// Mitsubishi GX Works2 project: Ex05   PLC: Q02/Q02H

PROGRAM MAIN
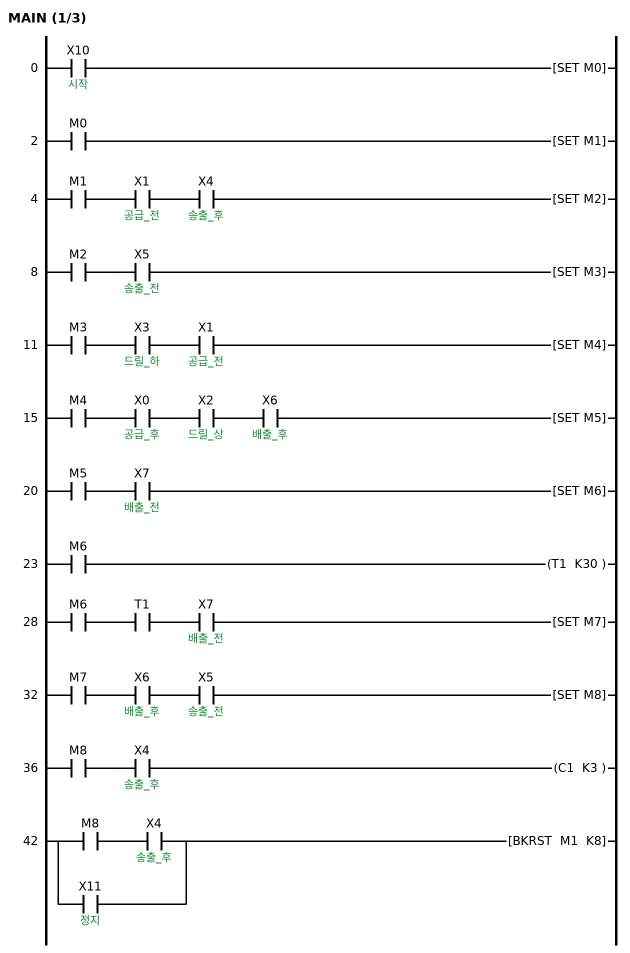
0     LD      X10  ; 시작
      SET     M0
2     LD      M0
      SET     M1
4     LD      M1
      AND     X1  ; 공급_전
      AND     X4  ; 송출_후
      SET     M2
8     LD      M2
      AND     X5  ; 송출_전
      SET     M3
11    LD      M3
      AND     X3  ; 드릴_하
      AND     X1  ; 공급_전
      SET     M4
15    LD      M4
      AND     X0  ; 공급_후
      AND     X2  ; 드릴_상
      AND     X6  ; 배출_후
      SET     M5
20    LD      M5
      AND     X7  ; 배출_전
      SET     M6
23    LD      M6
      OUT     T1 K30
28    LD      M6
      AND     T1
      AND     X7  ; 배출_전
      SET     M7
32    LD      M7
      AND     X6  ; 배출_후
      AND     X5  ; 송출_전
      SET     M8
36    LD      M8
      AND     X4  ; 송출_후
      OUT     C1 K3
42    LD      M8
      AND     X4  ; 송출_후
      OR      X11  ; 정지
      BKRST   M1 K8
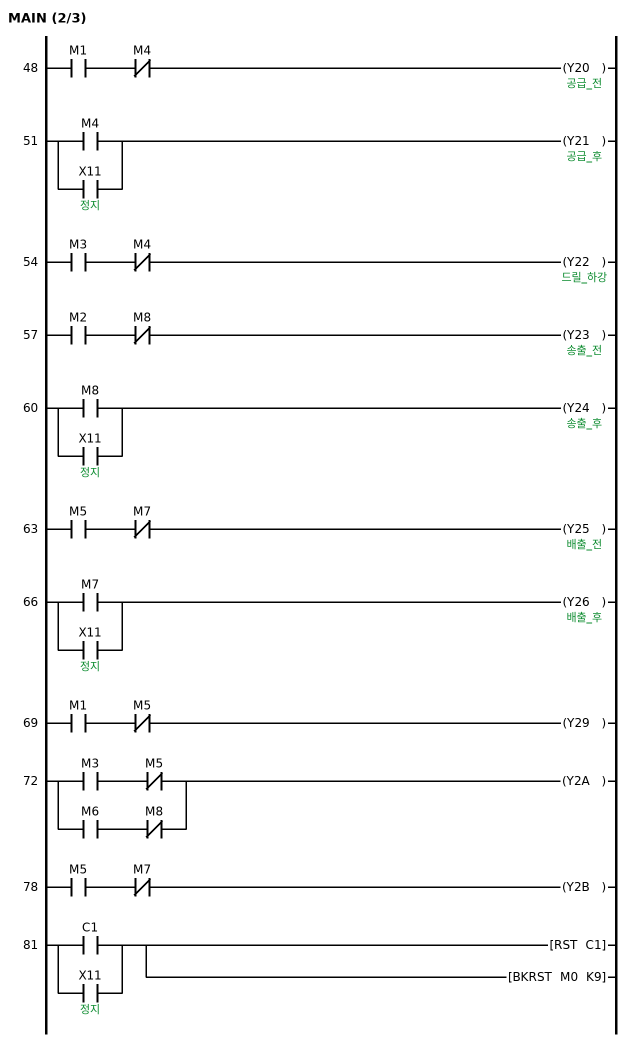
48    LD      M1
      ANI     M4
      OUT     Y20  ; 공급_전
51    LD      M4
      OR      X11  ; 정지
      OUT     Y21  ; 공급_후
54    LD      M3
      ANI     M4
      OUT     Y22  ; 드릴_하강
57    LD      M2
      ANI     M8
      OUT     Y23  ; 송출_전
60    LD      M8
      OR      X11  ; 정지
      OUT     Y24  ; 송출_후
63    LD      M5
      ANI     M7
      OUT     Y25  ; 배출_전
66    LD      M7
      OR      X11  ; 정지
      OUT     Y26  ; 배출_후
69    LD      M1
      ANI     M5
      OUT     Y29
72    LD      M3
      ANI     M5
      LD      M6
      ANI     M8
      ORB
      OUT     Y2A
78    LD      M5
      ANI     M7
      OUT     Y2B
81    LD      C1
      OR      X11  ; 정지
      RST     C1
      BKRST   M0 K9
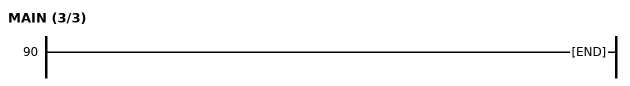
90    END
END_PROGRAM
